// TIA Portal V18 export
VAR_GLOBAL   // PLC tag table "Cabinet_2"
   Sz2_Button_LED_ST27_ST28 AT %Q1200.0 : Bool;
   Sz2_Button_LED_ST28_ST29 AT %Q1200.1 : Bool;
   Sz2_Button_LED_ST22_ST21 AT %Q1200.2 : Bool;
   Sz2_Button_LED_ST21_ST20 AT %Q1200.3 : Bool;
   Sz2_Button_LED_Centering_ST21 AT %Q1200.4 : Bool;
   Sz2_Button_LED_Centering_ST20 AT %Q1200.5 : Bool;
   "Reserved(25)" AT %Q1200.6 : Bool;
   "Reserved(26)" AT %Q1200.7 : Bool;
   Sz2_ST27_SenA AT %I1200.0 : Bool;
   Sz2_ST27_SenB AT %I1200.1 : Bool;
   Sz2_ST27_SenC AT %I1200.2 : Bool;
   Sz2_ST27_SenD AT %I1200.3 : Bool;
   Sz2_ST28_SenA AT %I1200.4 : Bool;
   Sz2_ST28_SenB AT %I1200.5 : Bool;
   Sz2_ST28_SenC AT %I1200.6 : Bool;
   Sz2_ST28_SenD AT %I1200.7 : Bool;
   Sz2_ST21_SenA AT %I1201.0 : Bool;
   Sz2_ST21_SenB AT %I1201.1 : Bool;
   Sz2_ST21_SenC AT %I1201.2 : Bool;
   Sz2_ST21_SenD AT %I1201.3 : Bool;
   Sz2_ST22_SenA AT %I1201.4 : Bool;
   Sz2_ST22_SenB AT %I1201.5 : Bool;
   Sz2_ST22_SenC AT %I1201.6 : Bool;
   Sz2_ST22_SenD AT %I1201.7 : Bool;
   Sz2_Button_ST27_ST28 AT %I1202.0 : Bool;
   Sz2_Button_ST28_ST29 AT %I1202.1 : Bool;
   Sz2_Button_ST22_ST21 AT %I1202.2 : Bool;
   Sz2_Button_ST21_ST20 AT %I1202.3 : Bool;
   Sz2_Button_Centering_ST21 AT %I1202.4 : Bool;
   Sz2_Button_Centering_ST20 AT %I1202.5 : Bool;
   "Reserved(27)" AT %I1202.6 : Bool;
   "Reserved(28)" AT %I1202.7 : Bool;
   Sz2_Safety_1_1 AT %I1250.0 : Bool;
   Sz2_Safety_1_2 AT %I1250.4 : Bool;
   "Reserved(29)" AT %I1250.1 : Bool;
   "Reserved(30)" AT %I1250.2 : Bool;
   "Reserved(31)" AT %I1250.3 : Bool;
   "Reserved(32)" AT %I1250.5 : Bool;
   "Reserved(33)" AT %I1250.6 : Bool;
   "Reserved(34)" AT %I1250.7 : Bool;
   "Reserved(35)" AT %I1251.0 : Bool;
   "Reserved(36)" AT %I1251.1 : Bool;
   "Reserved(37)" AT %I1251.2 : Bool;
   "Reserved(38)" AT %I1251.3 : Bool;
   "Reserved(39)" AT %I1251.4 : Bool;
   "Reserved(40)" AT %I1251.5 : Bool;
   "Reserved(41)" AT %I1251.6 : Bool;
   "Reserved(42)" AT %I1251.7 : Bool;
END_VAR
